// Block: FinalCut_PERS

DATA_BLOCK FinalCut_PERS
VERSION : 0.1
   NON_RETAIN
   VAR
      PersistentValues : udt_FinalCut_Pers;
   END_VAR

BEGIN
   // No initialization required
END_DATA_BLOCK
